% RSLogix 500 project Freezers Onsite - 17-4-07 - Before Changes.RSS, saved by version 7.00.00.19 %
PROJECT "UNTITLED"    % processor: SLC 500, 1747-L531 %

PROGRAM FILES
  LAD 2   14 rungs
  LAD 3   32 rungs
  LAD 4   57 rungs
  LAD 5   84 rungs
  LAD 6   10 rungs
  LAD 7   14 rungs
  LAD 8   20 rungs
  LAD 9, 10: only END

DATA FILES
  O0 OUTPUT  3 elements
  I1 INPUT  7 elements
  S2 STATUS  83 elements
  B3 BINARY  20 elements
  T4 TIMER  50 elements
  C5 COUNTER  1 elements
  R6 CONTROL  1 elements
  N7 INTEGER  40 elements
  F8 FLOAT  1 elements
  B16   10 elements
  N17   40 elements
  N18   30 elements
  B19   10 elements
  N20   60 elements
  T21   40 elements
  B40   20 elements
  N41   80 elements
  B42   10 elements

LADDER 2
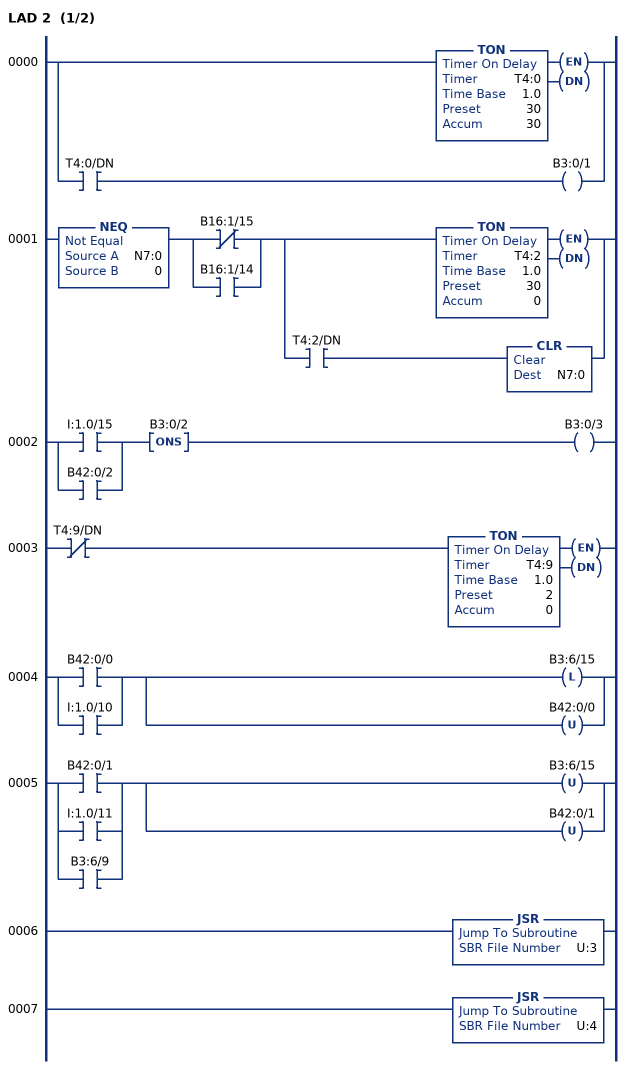
% Rung: 0 %
SOR BST TON T4:0 1.0 30 30 NXB XIC T4:0/DN OTE B3:0/1 BND EOR
% Rung: 1 %
SOR NEQ N7:0 0 BST XIO B16:1/15 NXB XIC B16:1/14 BND BST TON T4:2 1.0 30 0 NXB XIC T4:2/DN CLR N7:0 BND EOR
% Rung: 2 %
SOR BST XIC I:1.0/15 NXB XIC B42:0/2 BND OSR B3:0/2 OTE B3:0/3 EOR
% Rung: 3 %
SOR XIO T4:9/DN TON T4:9 1.0 2 0 EOR
% Rung: 4 %
SOR BST XIC B42:0/0 NXB XIC I:1.0/10 BND BST OTL B3:6/15 NXB OTU B42:0/0 BND EOR
% Rung: 5 %
SOR BST BST XIC B42:0/1 NXB XIC I:1.0/11 BND NXB XIC B3:6/9 BND BST OTU B3:6/15 NXB OTU B42:0/1 BND EOR
% Rung: 6 %
SOR JSR U:3 EOR
% Rung: 7 %
SOR JSR U:4 EOR

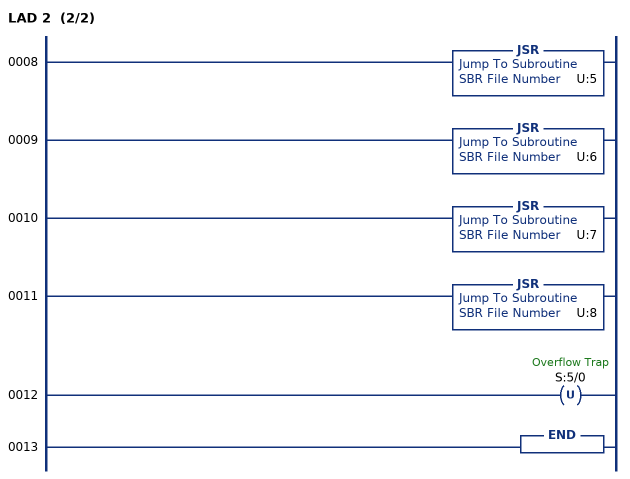
% Rung: 8 %
SOR JSR U:5 EOR
% Rung: 9 %
SOR JSR U:6 EOR
% Rung: 10 %
SOR JSR U:7 EOR
% Rung: 11 %
SOR JSR U:8 EOR
% Rung: 12 %
SOR OTU S:5/0 EOR
%   S:5/0  "Overflow Trap" %
% Rung: 13 %
SOR END EOR

LADDER 3
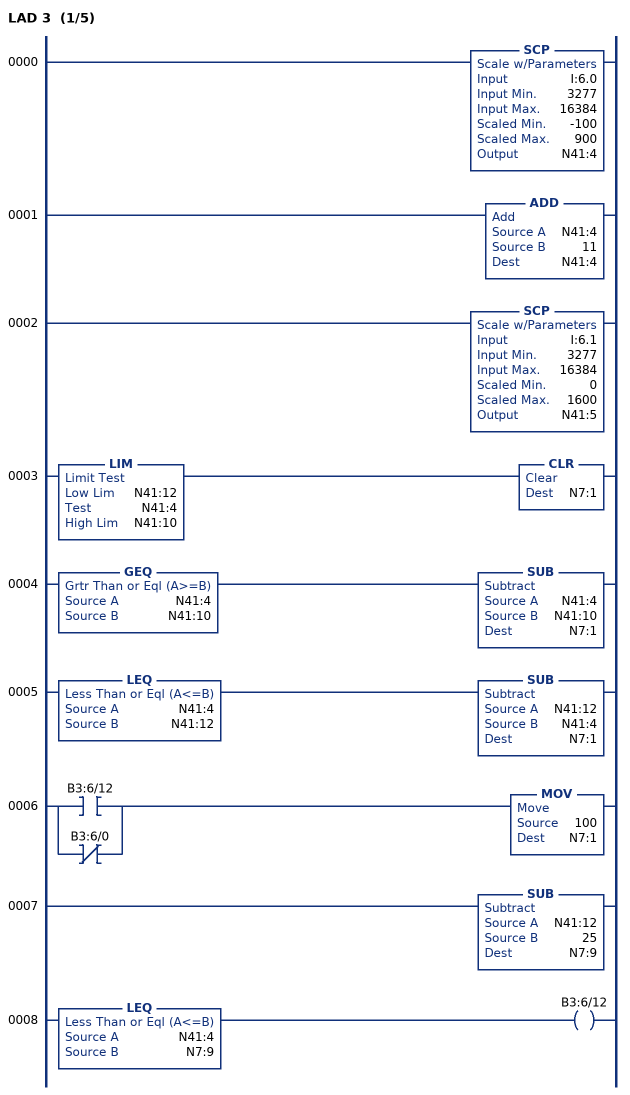
% Rung: 0 %
SOR SCP I:6.0 3277 16384 -100 900 N41:4 EOR
% Rung: 1 %
SOR ADD N41:4 11 N41:4 EOR
% Rung: 2 %
SOR SCP I:6.1 3277 16384 0 1600 N41:5 EOR
% Rung: 3 %
SOR LIM N41:12 N41:4 N41:10 CLR N7:1 EOR
% Rung: 4 %
SOR GEQ N41:4 N41:10 SUB N41:4 N41:10 N7:1 EOR
% Rung: 5 %
SOR LEQ N41:4 N41:12 SUB N41:12 N41:4 N7:1 EOR
% Rung: 6 %
SOR BST XIC B3:6/12 NXB XIO B3:6/0 BND MOV 100 N7:1 EOR
% Rung: 7 %
SOR SUB N41:12 25 N7:9 EOR
% Rung: 8 %
SOR LEQ N41:4 N7:9 OTE B3:6/12 EOR

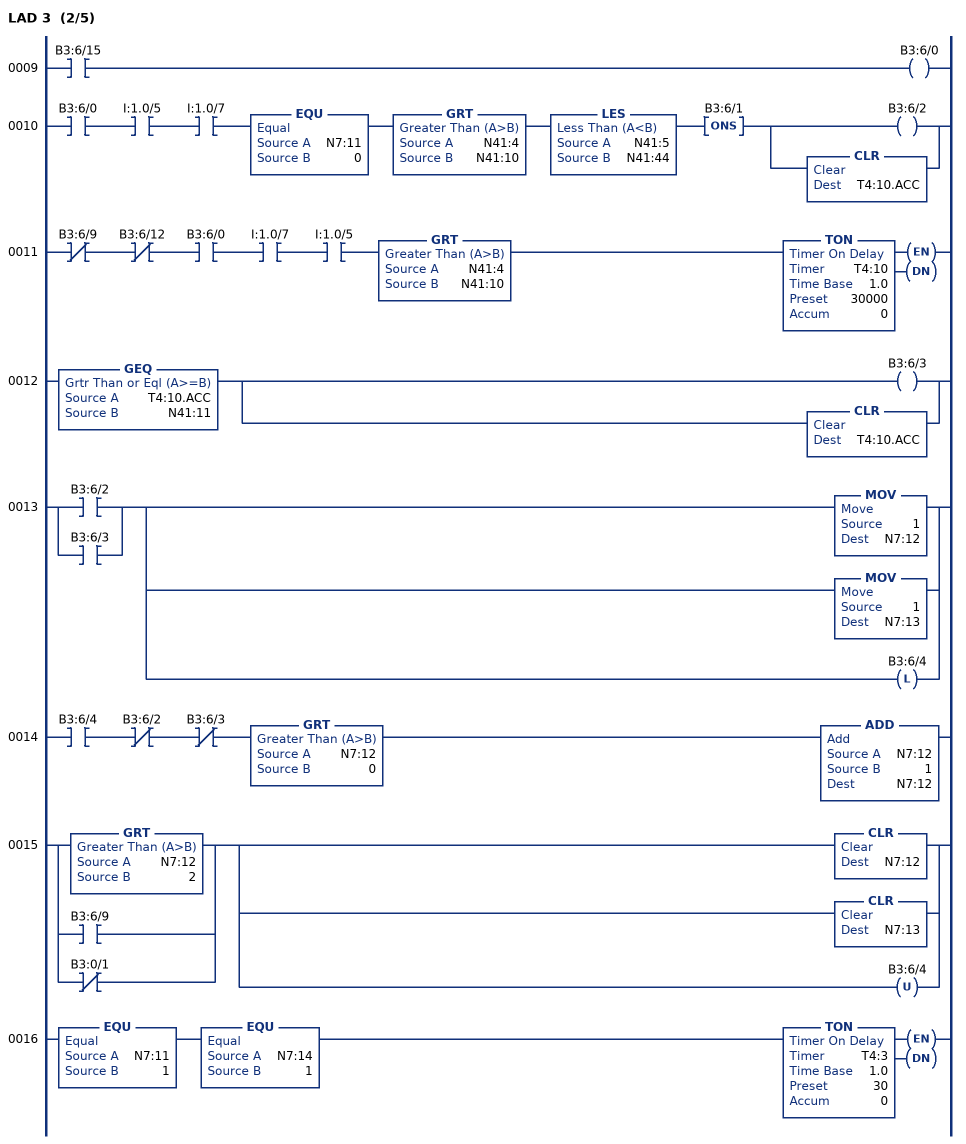
% Rung: 9 %
SOR XIC B3:6/15 OTE B3:6/0 EOR
% Rung: 10 %
SOR XIC B3:6/0 XIC I:1.0/5 XIC I:1.0/7 EQU N7:11 0 GRT N41:4 N41:10 LES N41:5 N41:44 OSR B3:6/1 BST OTE B3:6/2 NXB CLR T4:10.ACC BND EOR
% Rung: 11 %
SOR XIO B3:6/9 XIO B3:6/12 XIC B3:6/0 XIC I:1.0/7 XIC I:1.0/5 GRT N41:4 N41:10 TON T4:10 1.0 30000 0 EOR
% Rung: 12 %
SOR GEQ T4:10.ACC N41:11 BST OTE B3:6/3 NXB CLR T4:10.ACC BND EOR
% Rung: 13 %
SOR BST XIC B3:6/2 NXB XIC B3:6/3 BND BST MOV 1 N7:12 NXB MOV 1 N7:13 NXB OTL B3:6/4 BND EOR
% Rung: 14 %
SOR XIC B3:6/4 XIO B3:6/2 XIO B3:6/3 GRT N7:12 0 ADD N7:12 1 N7:12 EOR
% Rung: 15 %
SOR BST GRT N7:12 2 NXB XIC B3:6/9 NXB XIO B3:0/1 BND BST CLR N7:12 NXB CLR N7:13 NXB OTU B3:6/4 BND EOR
% Rung: 16 %
SOR EQU N7:11 1 EQU N7:14 1 TON T4:3 1.0 30 0 EOR

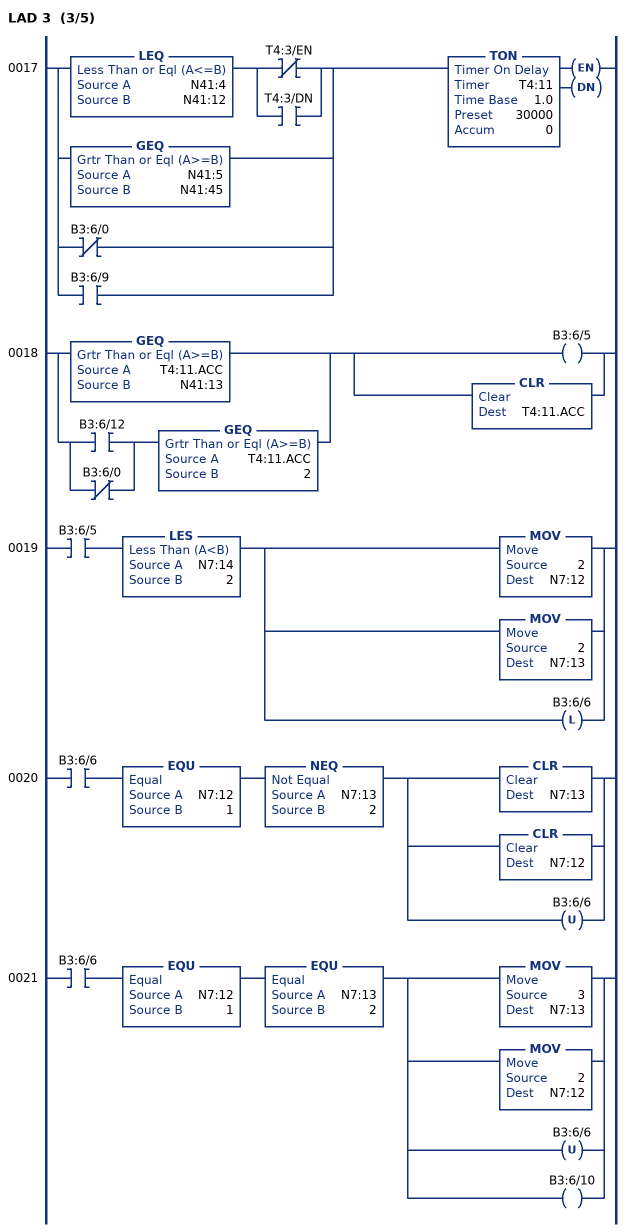
% Rung: 17 %
SOR BST LEQ N41:4 N41:12 BST XIO T4:3/EN NXB XIC T4:3/DN BND NXB GEQ N41:5 N41:45 NXB XIO B3:6/0 NXB XIC B3:6/9 BND TON T4:11 1.0 30000 0 EOR
% Rung: 18 %
SOR BST GEQ T4:11.ACC N41:13 NXB BST XIC B3:6/12 NXB XIO B3:6/0 BND GEQ T4:11.ACC 2 BND BST OTE B3:6/5 NXB CLR T4:11.ACC BND EOR
% Rung: 19 %
SOR XIC B3:6/5 LES N7:14 2 BST MOV 2 N7:12 NXB MOV 2 N7:13 NXB OTL B3:6/6 BND EOR
% Rung: 20 %
SOR XIC B3:6/6 EQU N7:12 1 NEQ N7:13 2 BST CLR N7:13 NXB CLR N7:12 NXB OTU B3:6/6 BND EOR
% Rung: 21 %
SOR XIC B3:6/6 EQU N7:12 1 EQU N7:13 2 BST MOV 3 N7:13 NXB MOV 2 N7:12 NXB OTU B3:6/6 NXB OTE B3:6/10 BND EOR

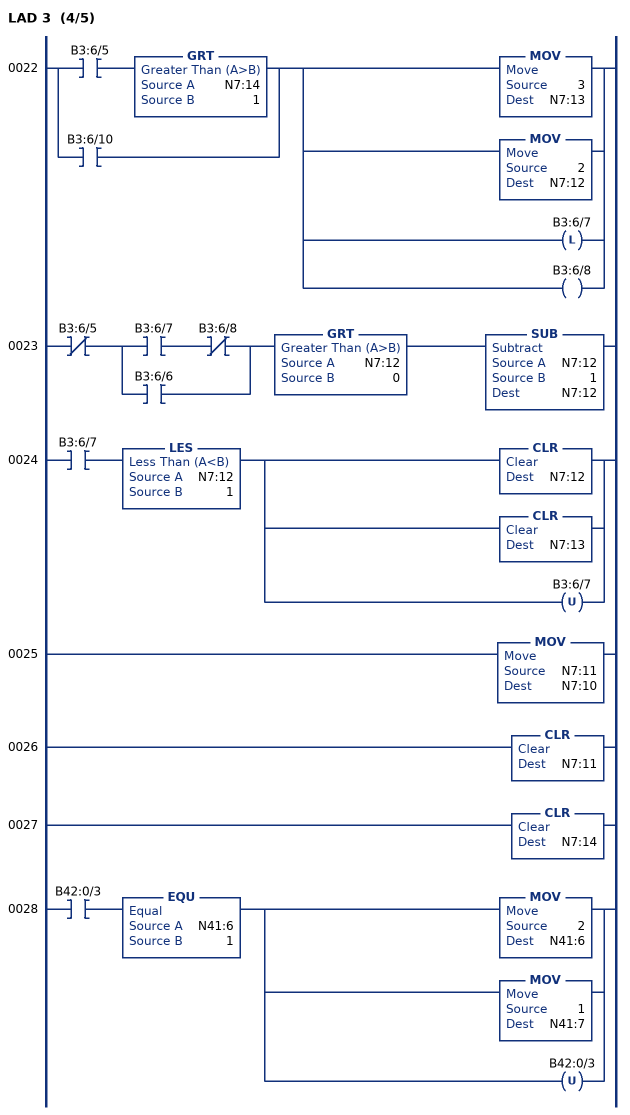
% Rung: 22 %
SOR BST XIC B3:6/5 GRT N7:14 1 NXB XIC B3:6/10 BND BST MOV 3 N7:13 NXB MOV 2 N7:12 NXB OTL B3:6/7 NXB OTE B3:6/8 BND EOR
% Rung: 23 %
SOR XIO B3:6/5 BST XIC B3:6/7 XIO B3:6/8 NXB XIC B3:6/6 BND GRT N7:12 0 SUB N7:12 1 N7:12 EOR
% Rung: 24 %
SOR XIC B3:6/7 LES N7:12 1 BST CLR N7:12 NXB CLR N7:13 NXB OTU B3:6/7 BND EOR
% Rung: 25 %
SOR MOV N7:11 N7:10 EOR
% Rung: 26 %
SOR CLR N7:11 EOR
% Rung: 27 %
SOR CLR N7:14 EOR
% Rung: 28 %
SOR XIC B42:0/3 EQU N41:6 1 BST MOV 2 N41:6 NXB MOV 1 N41:7 NXB OTU B42:0/3 BND EOR

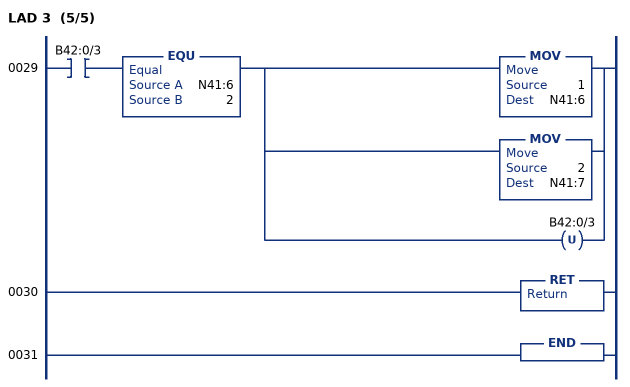
% Rung: 29 %
SOR XIC B42:0/3 EQU N41:6 2 BST MOV 1 N41:6 NXB MOV 2 N41:7 NXB OTU B42:0/3 BND EOR
% Rung: 30 %
SOR RET EOR
% Rung: 31 %
SOR END EOR

LADDER 4
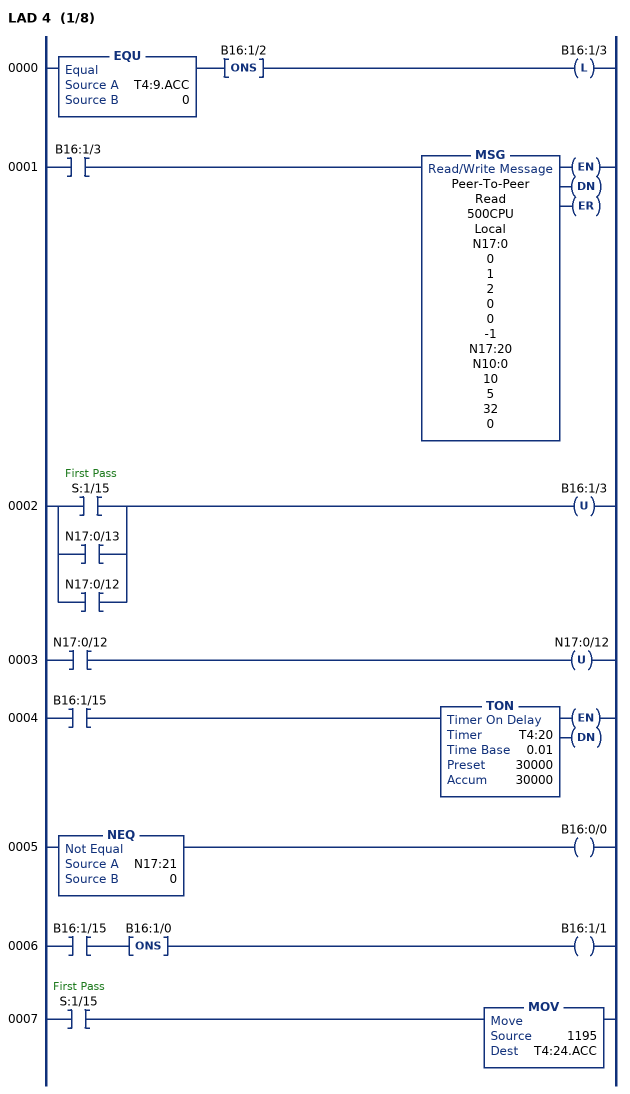
% Rung: 0 %
SOR EQU T4:9.ACC 0 OSR B16:1/2 OTL B16:1/3 EOR
% Rung: 1 %
SOR XIC B16:1/3 MSG Peer-To-Peer Read 500CPU Local N17:0 0 1 2 0 0 -1 N17:20 N10:0 10 5 32 0 EOR
%   MSG set-up: 500CPU Read | 5 | 10 | N10:0 | N17:20 | 0 | 2 | 2 | CLIENT | 0 | 0 %
% Rung: 2 %
SOR BST XIC S:1/15 NXB XIC N17:0/13 NXB XIC N17:0/12 BND OTU B16:1/3 EOR
%   S:1/15  "First Pass" %
% Rung: 3 %
SOR XIC N17:0/12 OTU N17:0/12 EOR
% Rung: 4 %
SOR XIC B16:1/15 TON T4:20 0.01 30000 30000 EOR
% Rung: 5 %
SOR NEQ N17:21 0 OTE B16:0/0 EOR
% Rung: 6 %
SOR XIC B16:1/15 OSR B16:1/0 OTE B16:1/1 EOR
% Rung: 7 %
SOR XIC S:1/15 MOV 1195 T4:24.ACC EOR
%   S:1/15  "First Pass" %

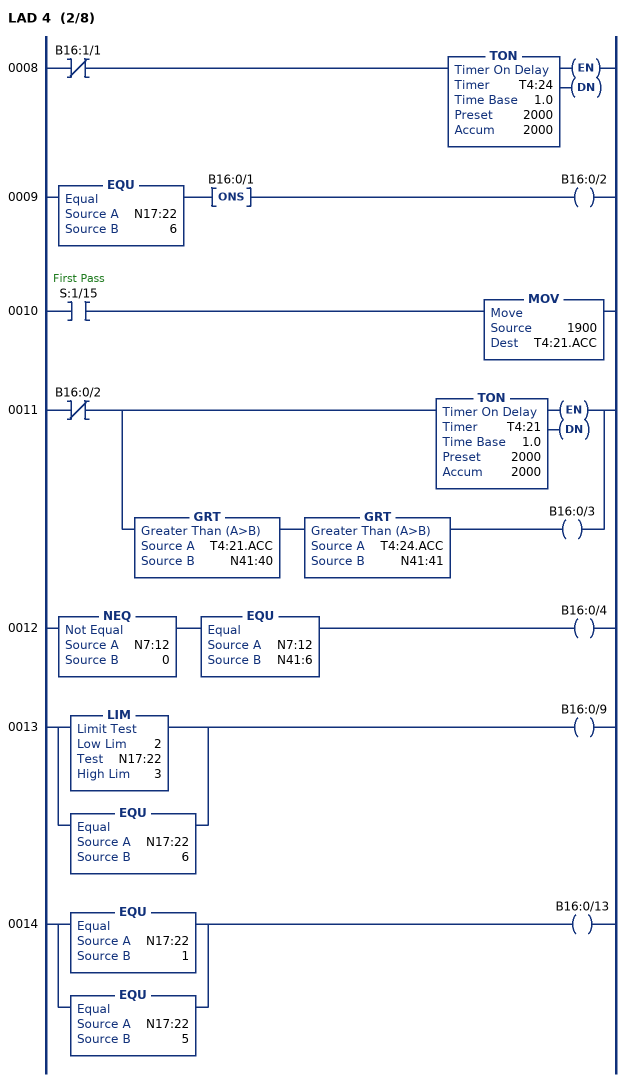
% Rung: 8 %
SOR XIO B16:1/1 TON T4:24 1.0 2000 2000 EOR
% Rung: 9 %
SOR EQU N17:22 6 OSR B16:0/1 OTE B16:0/2 EOR
% Rung: 10 %
SOR XIC S:1/15 MOV 1900 T4:21.ACC EOR
%   S:1/15  "First Pass" %
% Rung: 11 %
SOR XIO B16:0/2 BST TON T4:21 1.0 2000 2000 NXB GRT T4:21.ACC N41:40 GRT T4:24.ACC N41:41 OTE B16:0/3 BND EOR
% Rung: 12 %
SOR NEQ N7:12 0 EQU N7:12 N41:6 OTE B16:0/4 EOR
% Rung: 13 %
SOR BST LIM 2 N17:22 3 NXB EQU N17:22 6 BND OTE B16:0/9 EOR
% Rung: 14 %
SOR BST EQU N17:22 1 NXB EQU N17:22 5 BND OTE B16:0/13 EOR

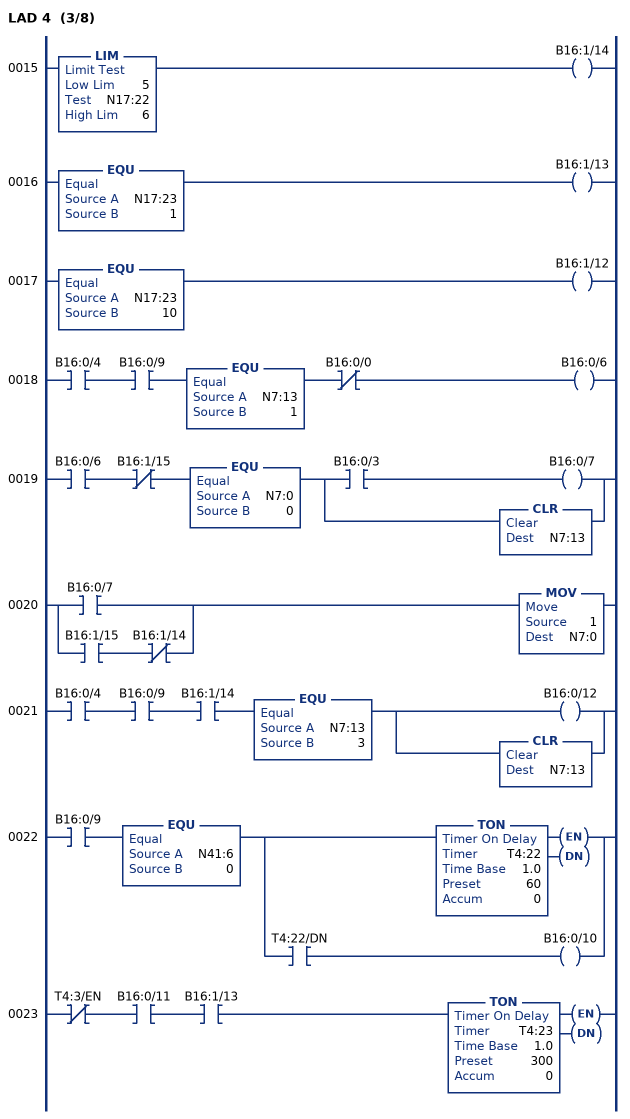
% Rung: 15 %
SOR LIM 5 N17:22 6 OTE B16:1/14 EOR
% Rung: 16 %
SOR EQU N17:23 1 OTE B16:1/13 EOR
% Rung: 17 %
SOR EQU N17:23 10 OTE B16:1/12 EOR
% Rung: 18 %
SOR XIC B16:0/4 XIC B16:0/9 EQU N7:13 1 XIO B16:0/0 OTE B16:0/6 EOR
% Rung: 19 %
SOR XIC B16:0/6 XIO B16:1/15 EQU N7:0 0 BST XIC B16:0/3 OTE B16:0/7 NXB CLR N7:13 BND EOR
% Rung: 20 %
SOR BST XIC B16:0/7 NXB XIC B16:1/15 XIO B16:1/14 BND MOV 1 N7:0 EOR
% Rung: 21 %
SOR XIC B16:0/4 XIC B16:0/9 XIC B16:1/14 EQU N7:13 3 BST OTE B16:0/12 NXB CLR N7:13 BND EOR
% Rung: 22 %
SOR XIC B16:0/9 EQU N41:6 0 BST TON T4:22 1.0 60 0 NXB XIC T4:22/DN OTE B16:0/10 BND EOR
% Rung: 23 %
SOR XIO T4:3/EN XIC B16:0/11 XIC B16:1/13 TON T4:23 1.0 300 0 EOR

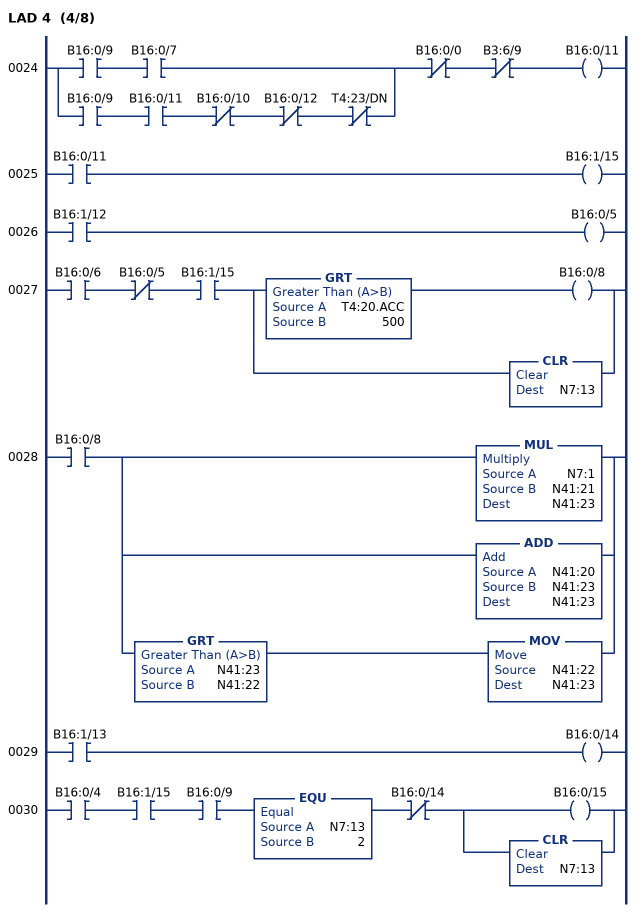
% Rung: 24 %
SOR BST XIC B16:0/9 XIC B16:0/7 NXB XIC B16:0/9 XIC B16:0/11 XIO B16:0/10 XIO B16:0/12 XIO T4:23/DN BND XIO B16:0/0 XIO B3:6/9 OTE B16:0/11 EOR
% Rung: 25 %
SOR XIC B16:0/11 OTE B16:1/15 EOR
% Rung: 26 %
SOR XIC B16:1/12 OTE B16:0/5 EOR
% Rung: 27 %
SOR XIC B16:0/6 XIO B16:0/5 XIC B16:1/15 BST GRT T4:20.ACC 500 OTE B16:0/8 NXB CLR N7:13 BND EOR
% Rung: 28 %
SOR XIC B16:0/8 BST MUL N7:1 N41:21 N41:23 NXB ADD N41:20 N41:23 N41:23 NXB GRT N41:23 N41:22 MOV N41:22 N41:23 BND EOR
% Rung: 29 %
SOR XIC B16:1/13 OTE B16:0/14 EOR
% Rung: 30 %
SOR XIC B16:0/4 XIC B16:1/15 XIC B16:0/9 EQU N7:13 2 XIO B16:0/14 BST OTE B16:0/15 NXB CLR N7:13 BND EOR

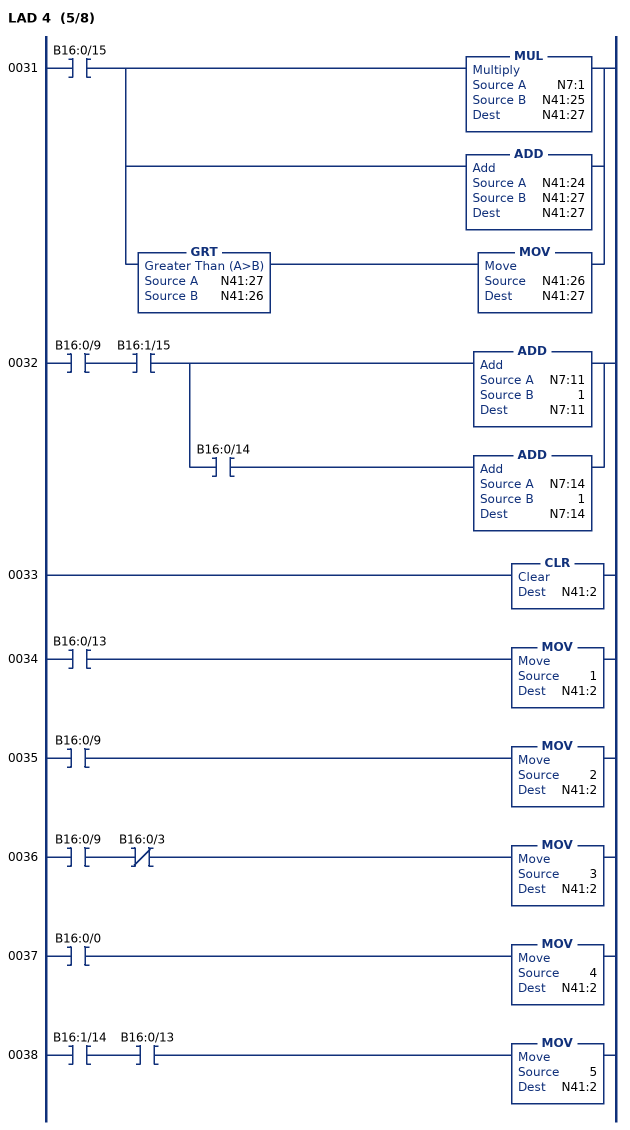
% Rung: 31 %
SOR XIC B16:0/15 BST MUL N7:1 N41:25 N41:27 NXB ADD N41:24 N41:27 N41:27 NXB GRT N41:27 N41:26 MOV N41:26 N41:27 BND EOR
% Rung: 32 %
SOR XIC B16:0/9 XIC B16:1/15 BST ADD N7:11 1 N7:11 NXB XIC B16:0/14 ADD N7:14 1 N7:14 BND EOR
% Rung: 33 %
SOR CLR N41:2 EOR
% Rung: 34 %
SOR XIC B16:0/13 MOV 1 N41:2 EOR
% Rung: 35 %
SOR XIC B16:0/9 MOV 2 N41:2 EOR
% Rung: 36 %
SOR XIC B16:0/9 XIO B16:0/3 MOV 3 N41:2 EOR
% Rung: 37 %
SOR XIC B16:0/0 MOV 4 N41:2 EOR
% Rung: 38 %
SOR XIC B16:1/14 XIC B16:0/13 MOV 5 N41:2 EOR

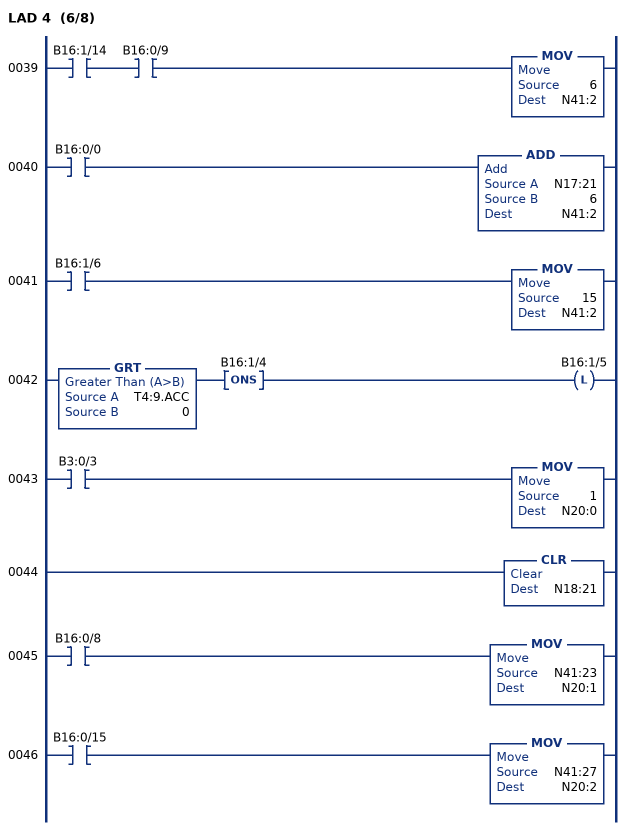
% Rung: 39 %
SOR XIC B16:1/14 XIC B16:0/9 MOV 6 N41:2 EOR
% Rung: 40 %
SOR XIC B16:0/0 ADD N17:21 6 N41:2 EOR
% Rung: 41 %
SOR XIC B16:1/6 MOV 15 N41:2 EOR
% Rung: 42 %
SOR GRT T4:9.ACC 0 OSR B16:1/4 OTL B16:1/5 EOR
% Rung: 43 %
SOR XIC B3:0/3 MOV 1 N20:0 EOR
% Rung: 44 %
SOR CLR N18:21 EOR
% Rung: 45 %
SOR XIC B16:0/8 MOV N41:23 N20:1 EOR
% Rung: 46 %
SOR XIC B16:0/15 MOV N41:27 N20:2 EOR

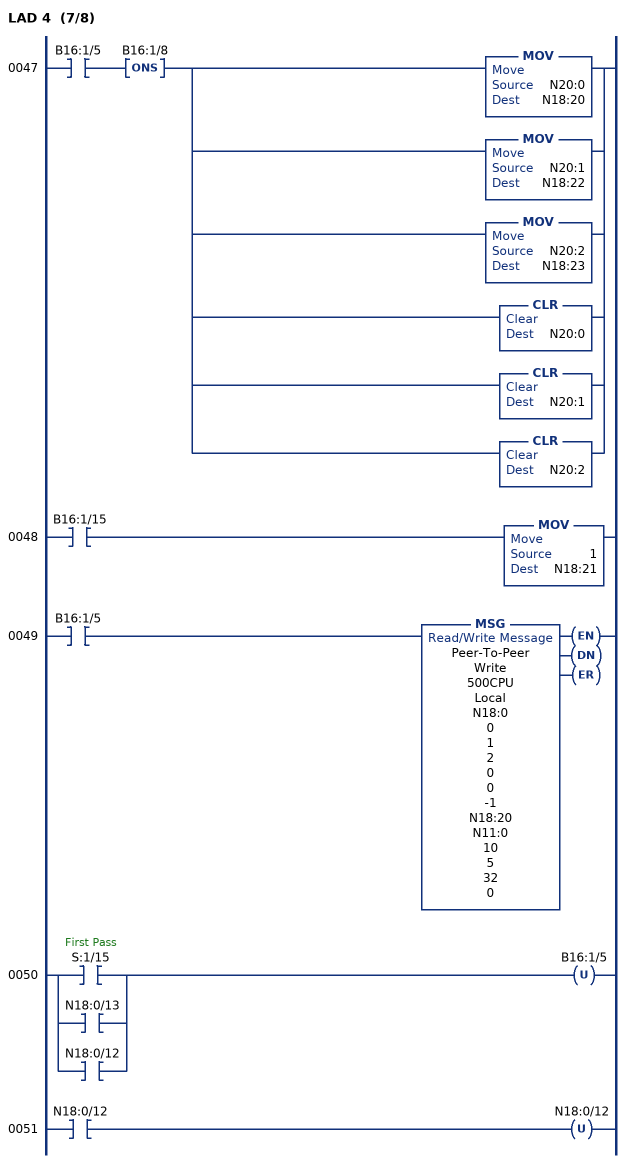
% Rung: 47 %
SOR XIC B16:1/5 OSR B16:1/8 BST MOV N20:0 N18:20 NXB MOV N20:1 N18:22 NXB MOV N20:2 N18:23 NXB CLR N20:0 NXB CLR N20:1 NXB CLR N20:2 BND EOR
% Rung: 48 %
SOR XIC B16:1/15 MOV 1 N18:21 EOR
% Rung: 49 %
SOR XIC B16:1/5 MSG Peer-To-Peer Write 500CPU Local N18:0 0 1 2 0 0 -1 N18:20 N11:0 10 5 32 0 EOR
%   MSG set-up: 500CPU Write | 5 | 10 | N11:0 | N18:20 | 0 | 2 | 2 | CLIENT | 0 | 0 %
% Rung: 50 %
SOR BST XIC S:1/15 NXB XIC N18:0/13 NXB XIC N18:0/12 BND OTU B16:1/5 EOR
%   S:1/15  "First Pass" %
% Rung: 51 %
SOR XIC N18:0/12 OTU N18:0/12 EOR

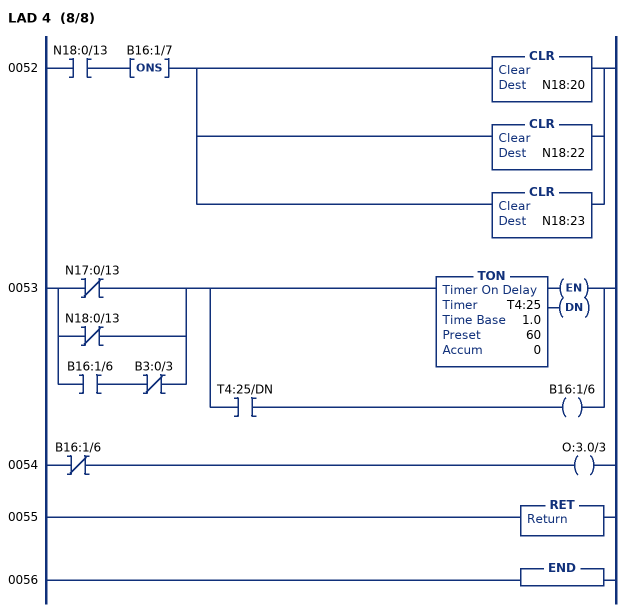
% Rung: 52 %
SOR XIC N18:0/13 OSR B16:1/7 BST CLR N18:20 NXB CLR N18:22 NXB CLR N18:23 BND EOR
% Rung: 53 %
SOR BST XIO N17:0/13 NXB XIO N18:0/13 NXB XIC B16:1/6 XIO B3:0/3 BND BST TON T4:25 1.0 60 0 NXB XIC T4:25/DN OTE B16:1/6 BND EOR
% Rung: 54 %
SOR XIO B16:1/6 OTE O:3.0/3 EOR
% Rung: 55 %
SOR RET EOR
% Rung: 56 %
SOR END EOR

LADDER 5
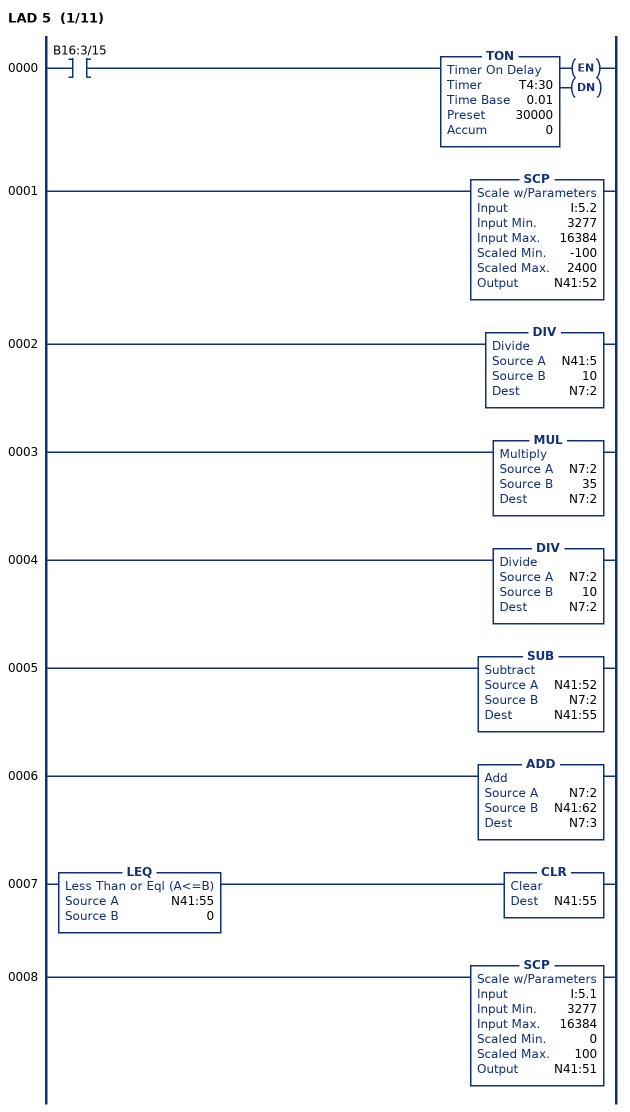
% Rung: 0 %
SOR XIC B16:3/15 TON T4:30 0.01 30000 0 EOR
% Rung: 1 %
SOR SCP I:5.2 3277 16384 -100 2400 N41:52 EOR
% Rung: 2 %
SOR DIV N41:5 10 N7:2 EOR
% Rung: 3 %
SOR MUL N7:2 35 N7:2 EOR
% Rung: 4 %
SOR DIV N7:2 10 N7:2 EOR
% Rung: 5 %
SOR SUB N41:52 N7:2 N41:55 EOR
% Rung: 6 %
SOR ADD N7:2 N41:62 N7:3 EOR
% Rung: 7 %
SOR LEQ N41:55 0 CLR N41:55 EOR
% Rung: 8 %
SOR SCP I:5.1 3277 16384 0 100 N41:51 EOR

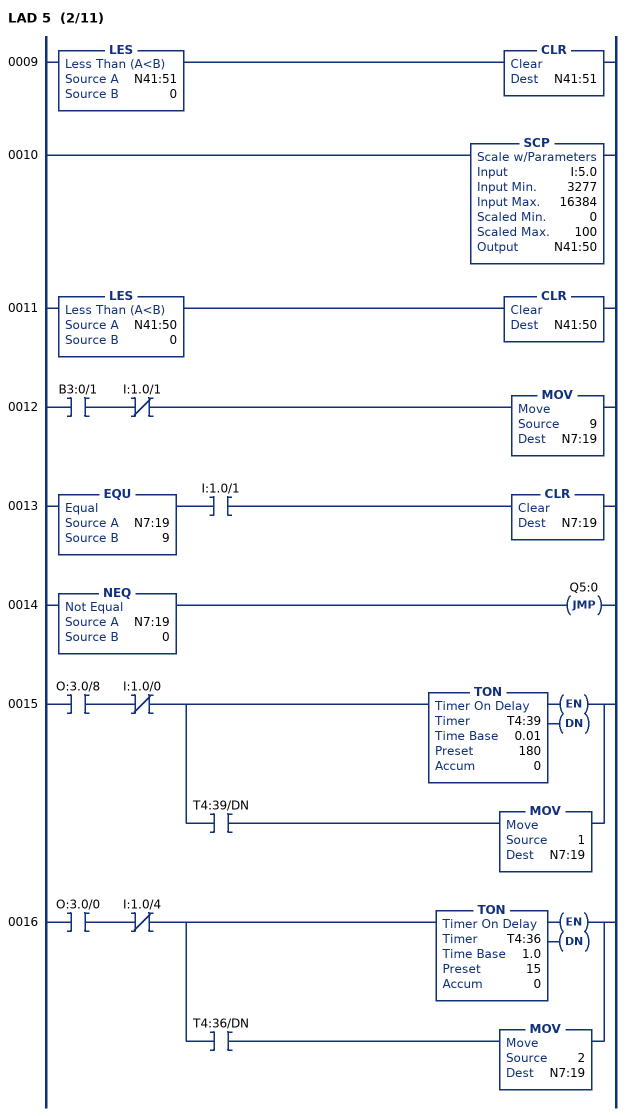
% Rung: 9 %
SOR LES N41:51 0 CLR N41:51 EOR
% Rung: 10 %
SOR SCP I:5.0 3277 16384 0 100 N41:50 EOR
% Rung: 11 %
SOR LES N41:50 0 CLR N41:50 EOR
% Rung: 12 %
SOR XIC B3:0/1 XIO I:1.0/1 MOV 9 N7:19 EOR
% Rung: 13 %
SOR EQU N7:19 9 XIC I:1.0/1 CLR N7:19 EOR
% Rung: 14 %
SOR NEQ N7:19 0 JMP Q5:0 EOR
% Rung: 15 %
SOR XIC O:3.0/8 XIO I:1.0/0 BST TON T4:39 0.01 180 0 NXB XIC T4:39/DN MOV 1 N7:19 BND EOR
% Rung: 16 %
SOR XIC O:3.0/0 XIO I:1.0/4 BST TON T4:36 1.0 15 0 NXB XIC T4:36/DN MOV 2 N7:19 BND EOR

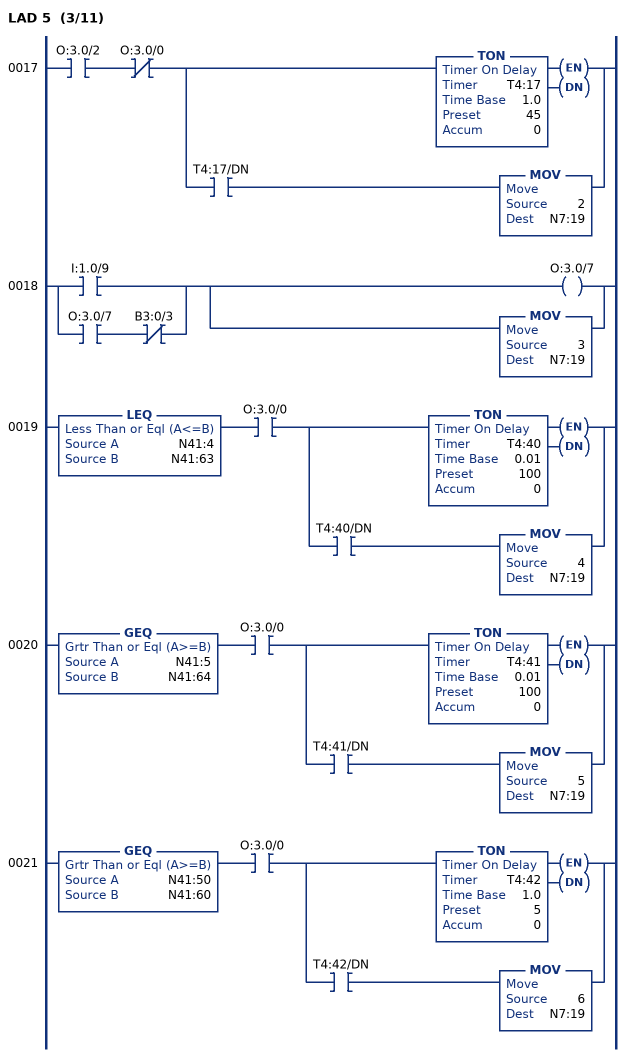
% Rung: 17 %
SOR XIC O:3.0/2 XIO O:3.0/0 BST TON T4:17 1.0 45 0 NXB XIC T4:17/DN MOV 2 N7:19 BND EOR
% Rung: 18 %
SOR BST XIC I:1.0/9 NXB XIC O:3.0/7 XIO B3:0/3 BND BST OTE O:3.0/7 NXB MOV 3 N7:19 BND EOR
% Rung: 19 %
SOR LEQ N41:4 N41:63 XIC O:3.0/0 BST TON T4:40 0.01 100 0 NXB XIC T4:40/DN MOV 4 N7:19 BND EOR
% Rung: 20 %
SOR GEQ N41:5 N41:64 XIC O:3.0/0 BST TON T4:41 0.01 100 0 NXB XIC T4:41/DN MOV 5 N7:19 BND EOR
% Rung: 21 %
SOR GEQ N41:50 N41:60 XIC O:3.0/0 BST TON T4:42 1.0 5 0 NXB XIC T4:42/DN MOV 6 N7:19 BND EOR

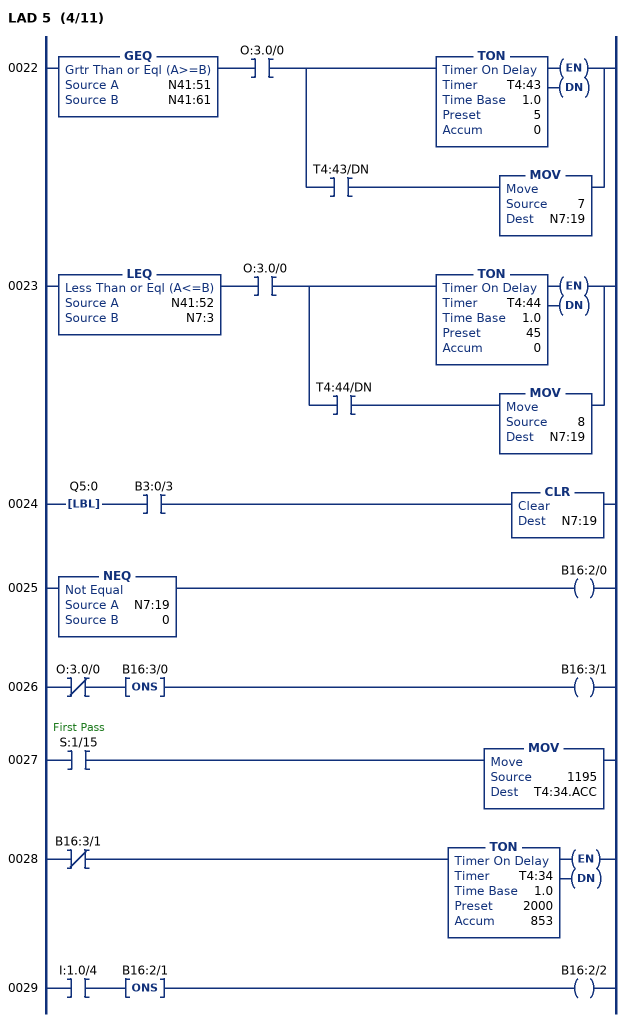
% Rung: 22 %
SOR GEQ N41:51 N41:61 XIC O:3.0/0 BST TON T4:43 1.0 5 0 NXB XIC T4:43/DN MOV 7 N7:19 BND EOR
% Rung: 23 %
SOR LEQ N41:52 N7:3 XIC O:3.0/0 BST TON T4:44 1.0 45 0 NXB XIC T4:44/DN MOV 8 N7:19 BND EOR
% Rung: 24 %
SOR LBL Q5:0 XIC B3:0/3 CLR N7:19 EOR
% Rung: 25 %
SOR NEQ N7:19 0 OTE B16:2/0 EOR
% Rung: 26 %
SOR XIO O:3.0/0 OSR B16:3/0 OTE B16:3/1 EOR
% Rung: 27 %
SOR XIC S:1/15 MOV 1195 T4:34.ACC EOR
%   S:1/15  "First Pass" %
% Rung: 28 %
SOR XIO B16:3/1 TON T4:34 1.0 2000 853 EOR
% Rung: 29 %
SOR XIC I:1.0/4 OSR B16:2/1 OTE B16:2/2 EOR

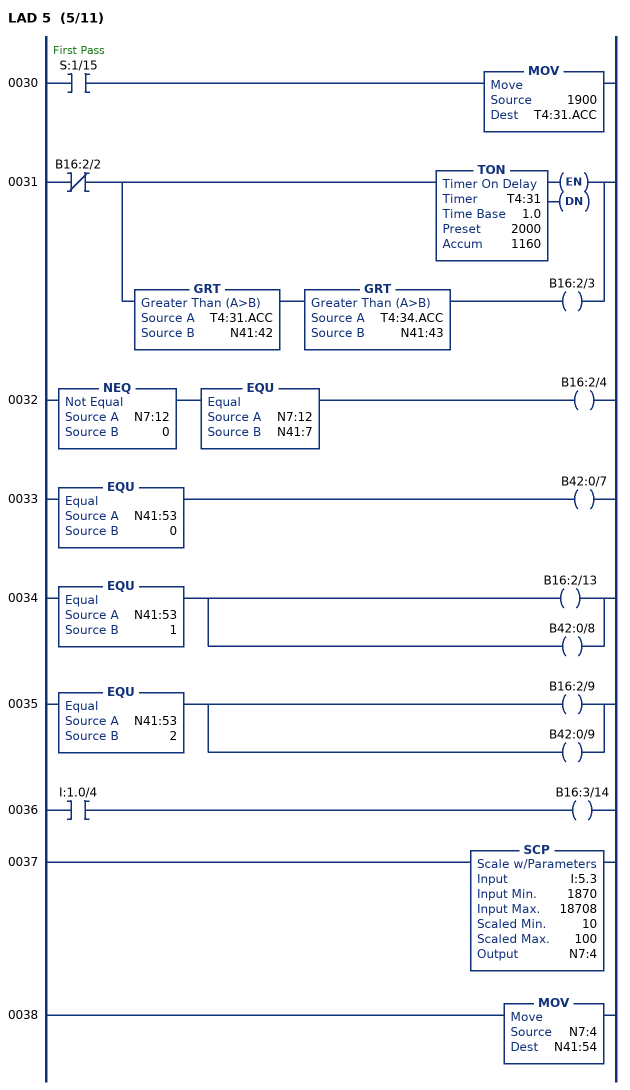
% Rung: 30 %
SOR XIC S:1/15 MOV 1900 T4:31.ACC EOR
%   S:1/15  "First Pass" %
% Rung: 31 %
SOR XIO B16:2/2 BST TON T4:31 1.0 2000 1160 NXB GRT T4:31.ACC N41:42 GRT T4:34.ACC N41:43 OTE B16:2/3 BND EOR
% Rung: 32 %
SOR NEQ N7:12 0 EQU N7:12 N41:7 OTE B16:2/4 EOR
% Rung: 33 %
SOR EQU N41:53 0 OTE B42:0/7 EOR
% Rung: 34 %
SOR EQU N41:53 1 BST OTE B16:2/13 NXB OTE B42:0/8 BND EOR
% Rung: 35 %
SOR EQU N41:53 2 BST OTE B16:2/9 NXB OTE B42:0/9 BND EOR
% Rung: 36 %
SOR XIC I:1.0/4 OTE B16:3/14 EOR
% Rung: 37 %
SOR SCP I:5.3 1870 18708 10 100 N7:4 EOR
% Rung: 38 %
SOR MOV N7:4 N41:54 EOR

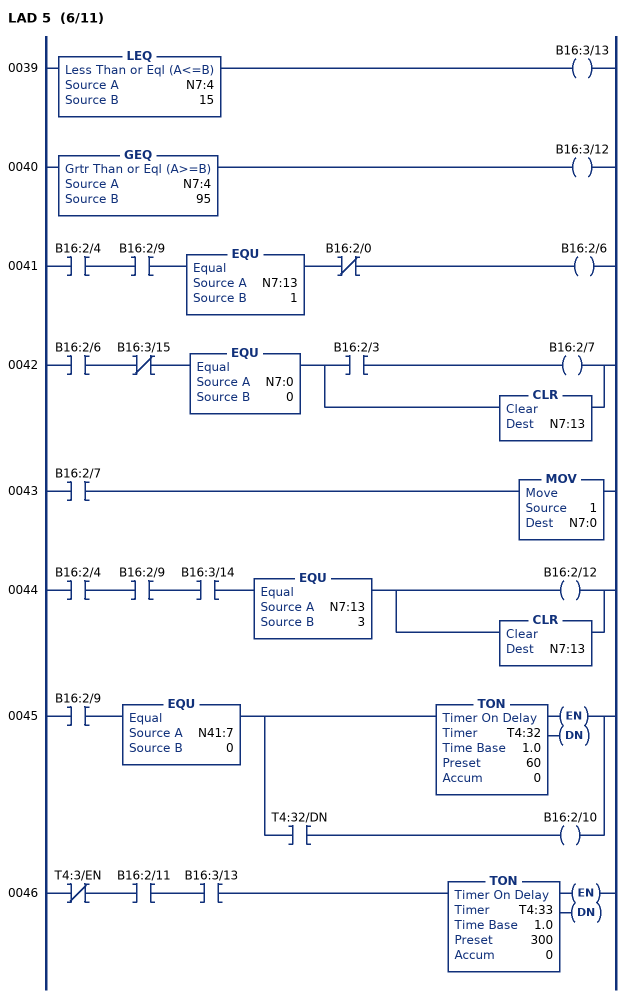
% Rung: 39 %
SOR LEQ N7:4 15 OTE B16:3/13 EOR
% Rung: 40 %
SOR GEQ N7:4 95 OTE B16:3/12 EOR
% Rung: 41 %
SOR XIC B16:2/4 XIC B16:2/9 EQU N7:13 1 XIO B16:2/0 OTE B16:2/6 EOR
% Rung: 42 %
SOR XIC B16:2/6 XIO B16:3/15 EQU N7:0 0 BST XIC B16:2/3 OTE B16:2/7 NXB CLR N7:13 BND EOR
% Rung: 43 %
SOR XIC B16:2/7 MOV 1 N7:0 EOR
% Rung: 44 %
SOR XIC B16:2/4 XIC B16:2/9 XIC B16:3/14 EQU N7:13 3 BST OTE B16:2/12 NXB CLR N7:13 BND EOR
% Rung: 45 %
SOR XIC B16:2/9 EQU N41:7 0 BST TON T4:32 1.0 60 0 NXB XIC T4:32/DN OTE B16:2/10 BND EOR
% Rung: 46 %
SOR XIO T4:3/EN XIC B16:2/11 XIC B16:3/13 TON T4:33 1.0 300 0 EOR

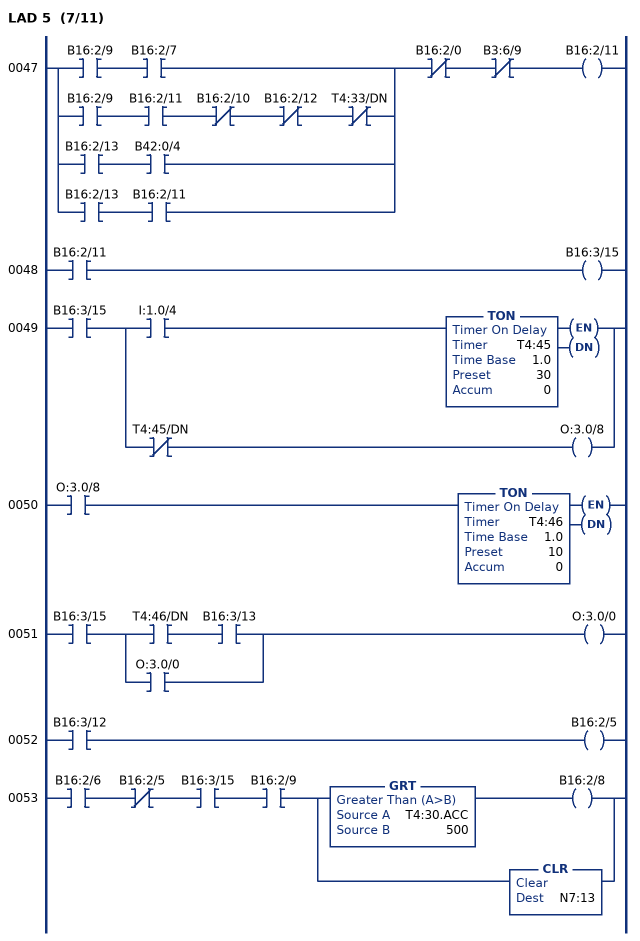
% Rung: 47 %
SOR BST XIC B16:2/9 XIC B16:2/7 NXB XIC B16:2/9 XIC B16:2/11 XIO B16:2/10 XIO B16:2/12 XIO T4:33/DN NXB XIC B16:2/13 XIC B42:0/4 NXB XIC B16:2/13 XIC B16:2/11 BND XIO B16:2/0 XIO B3:6/9 OTE B16:2/11 EOR
% Rung: 48 %
SOR XIC B16:2/11 OTE B16:3/15 EOR
% Rung: 49 %
SOR XIC B16:3/15 BST XIC I:1.0/4 TON T4:45 1.0 30 0 NXB XIO T4:45/DN OTE O:3.0/8 BND EOR
% Rung: 50 %
SOR XIC O:3.0/8 TON T4:46 1.0 10 0 EOR
% Rung: 51 %
SOR XIC B16:3/15 BST XIC T4:46/DN XIC B16:3/13 NXB XIC O:3.0/0 BND OTE O:3.0/0 EOR
% Rung: 52 %
SOR XIC B16:3/12 OTE B16:2/5 EOR
% Rung: 53 %
SOR XIC B16:2/6 XIO B16:2/5 XIC B16:3/15 XIC B16:2/9 BST GRT T4:30.ACC 500 OTE B16:2/8 NXB CLR N7:13 BND EOR

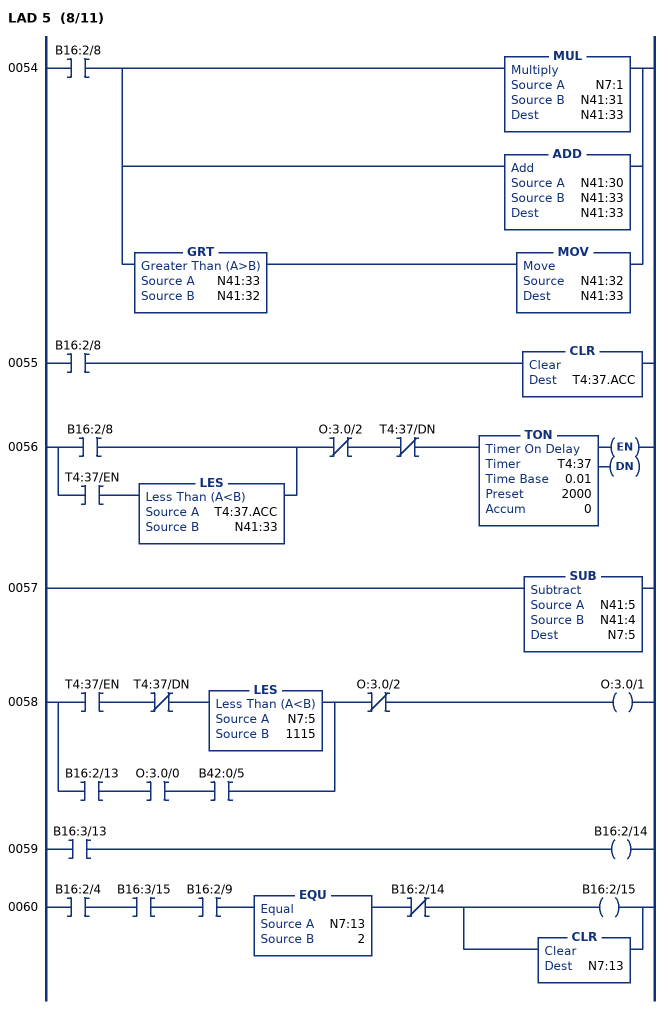
% Rung: 54 %
SOR XIC B16:2/8 BST MUL N7:1 N41:31 N41:33 NXB ADD N41:30 N41:33 N41:33 NXB GRT N41:33 N41:32 MOV N41:32 N41:33 BND EOR
% Rung: 55 %
SOR XIC B16:2/8 CLR T4:37.ACC EOR
% Rung: 56 %
SOR BST XIC B16:2/8 NXB XIC T4:37/EN LES T4:37.ACC N41:33 BND XIO O:3.0/2 XIO T4:37/DN TON T4:37 0.01 2000 0 EOR
% Rung: 57 %
SOR SUB N41:5 N41:4 N7:5 EOR
% Rung: 58 %
SOR BST XIC T4:37/EN XIO T4:37/DN LES N7:5 1115 NXB XIC B16:2/13 XIC O:3.0/0 XIC B42:0/5 BND XIO O:3.0/2 OTE O:3.0/1 EOR
% Rung: 59 %
SOR XIC B16:3/13 OTE B16:2/14 EOR
% Rung: 60 %
SOR XIC B16:2/4 XIC B16:3/15 XIC B16:2/9 EQU N7:13 2 XIO B16:2/14 BST OTE B16:2/15 NXB CLR N7:13 BND EOR

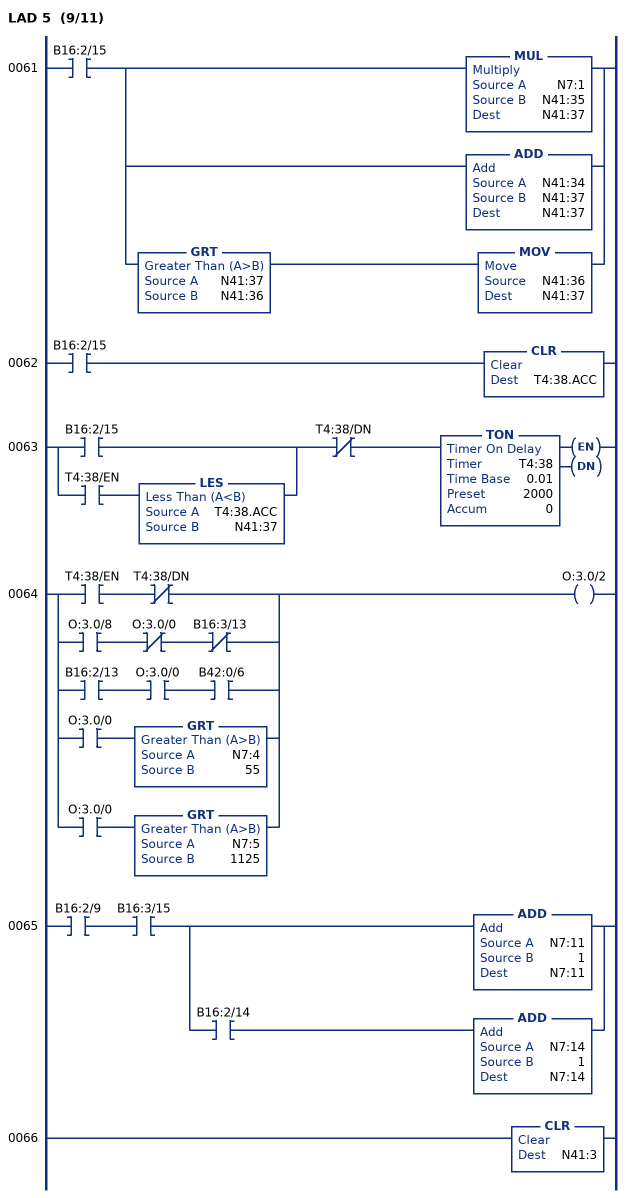
% Rung: 61 %
SOR XIC B16:2/15 BST MUL N7:1 N41:35 N41:37 NXB ADD N41:34 N41:37 N41:37 NXB GRT N41:37 N41:36 MOV N41:36 N41:37 BND EOR
% Rung: 62 %
SOR XIC B16:2/15 CLR T4:38.ACC EOR
% Rung: 63 %
SOR BST XIC B16:2/15 NXB XIC T4:38/EN LES T4:38.ACC N41:37 BND XIO T4:38/DN TON T4:38 0.01 2000 0 EOR
% Rung: 64 %
SOR BST XIC T4:38/EN XIO T4:38/DN NXB XIC O:3.0/8 XIO O:3.0/0 XIO B16:3/13 NXB XIC B16:2/13 XIC O:3.0/0 XIC B42:0/6 NXB XIC O:3.0/0 GRT N7:4 55 NXB XIC O:3.0/0 GRT N7:5 1125 BND OTE O:3.0/2 EOR
% Rung: 65 %
SOR XIC B16:2/9 XIC B16:3/15 BST ADD N7:11 1 N7:11 NXB XIC B16:2/14 ADD N7:14 1 N7:14 BND EOR
% Rung: 66 %
SOR CLR N41:3 EOR

